// TIA Portal V17 export
// export: Created 2022-11-28T05:31:20.721325Z, ExportSetting WithDefaults, DisplayName Totally Integrated Automation Portal, DisplayVersion V17, DisplayName TIA Portal Openness, DisplayVersion V17, DisplayName TIA Portal Version Control Interface, DisplayVersion V17, DisplayName STEP 7 Professional, DisplayVersion V17, DisplayName STEP 7 Safety, DisplayVersion V17, DisplayName WinCC Professional, DisplayVersion V17
FUNCTION_BLOCK "FB_Sorting"   // FB1, LAD
{ S7_Optimized_Access := 'TRUE' }
VERSION : 0.1
// stored: AutoNumber true, IsIECCheckEnabled false, IsRetainMemResEnabled false, MemoryReserve 100, SetENOAutomatically false, UDAEnableTagReadback false
   VAR_INPUT
      Color : Int;
   END_VAR
   VAR
      "Step" : Int;
      IEC_Timer_Rojo { S7_SetPoint := 'True'} : TON_TIME;
      IEC_Timer_Eject { S7_SetPoint := 'True'} : TON_TIME;
      Detener_Banda { S7_SetPoint := 'True'} : TOF_TIME;
      Sensor_reading { S7_SetPoint := 'True'} : Int;
      IEC_Timer_ReadSensor { S7_SetPoint := 'True'} : TON_TIME;
      Conveyor0 { S7_SetPoint := 'True'} : Bool;
      Conveyor1 { S7_SetPoint := 'True'} : Bool;
      LapseEject : Time;
   END_VAR
   VAR CONSTANT
      LapseEjectWhite : Time := T#400ms;
      LapseEjectRed : Time := T#1400ms;
      LapseejectBlue : Time := T#2400ms;
   END_VAR
   VAR_TEMP   // added for the SCL form of the ladder/FBD networks
      _w1 : Bool;
   END_VAR
BEGIN

REGION Network 1
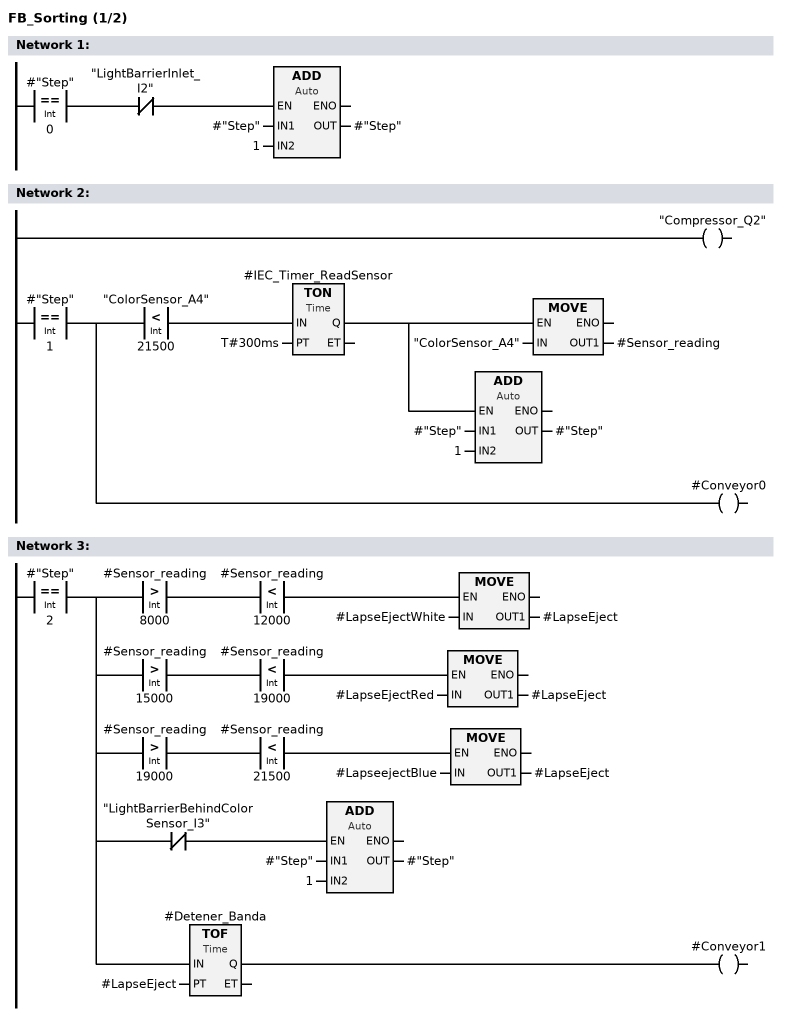
   RUNG wire#powerrail
      { S7_Templates := "SrcType := Int" } EQ_Contact(in1 := #"Step", in2 := 0)
      I_Contact( "LightBarrierInlet_I2" )
      Add(in1 := #"Step", in2 := 1, out => #"Step")
   END_RUNG
   // the same network as SCL:
   IF (#"Step" = 0) AND NOT "LightBarrierInlet_I2" THEN #"Step" := #"Step" + 1; END_IF;
END_REGION

REGION Network 2
   RUNG wire#powerrail
      Coil( "Compressor_Q2" )
   END_RUNG
   RUNG wire#powerrail
      { S7_Templates := "SrcType := Int" } EQ_Contact(in1 := #"Step", in2 := 1)
      wire#w1
      { S7_Templates := "SrcType := Int" } LT_Contact(in1 := "ColorSensor_A4", in2 := 21500)
      { S7_Templates := "time_type := Time" } #IEC_Timer_ReadSensor.TON(pt := T#300ms, et =>)
      wire#w2
      Move(in := "ColorSensor_A4", out1 => #Sensor_reading)
   END_RUNG
   RUNG wire#w2
      Add(in1 := #"Step", in2 := 1, out => #"Step")
   END_RUNG
   RUNG wire#w1
      Coil( #Conveyor0 )
   END_RUNG
   // the same network as SCL:
   "Compressor_Q2" := TRUE;
   #_w1 := #"Step" = 1;
   #IEC_Timer_ReadSensor(IN := #_w1 AND ("ColorSensor_A4" < 21500), PT := T#300ms);   // TON
   IF #IEC_Timer_ReadSensor.Q THEN
       #Sensor_reading := "ColorSensor_A4";
       #"Step" := #"Step" + 1;
   END_IF;
   #Conveyor0 := #_w1;
END_REGION

REGION Network 3
   RUNG wire#powerrail
      { S7_Templates := "SrcType := Int" } EQ_Contact(in1 := #"Step", in2 := 2)
      wire#w1
      { S7_Templates := "SrcType := Int" } GT_Contact(in1 := #Sensor_reading, in2 := 8000)
      { S7_Templates := "SrcType := Int" } LT_Contact(in1 := #Sensor_reading, in2 := 12000)
      Move(in := #LapseEjectWhite, out1 => #LapseEject)
   END_RUNG
   RUNG wire#w1
      { S7_Templates := "SrcType := Int" } GT_Contact(in1 := #Sensor_reading, in2 := 15000)
      { S7_Templates := "SrcType := Int" } LT_Contact(in1 := #Sensor_reading, in2 := 19000)
      Move(in := #LapseEjectRed, out1 => #LapseEject)
   END_RUNG
   RUNG wire#w1
      { S7_Templates := "SrcType := Int" } GT_Contact(in1 := #Sensor_reading, in2 := 19000)
      { S7_Templates := "SrcType := Int" } LT_Contact(in1 := #Sensor_reading, in2 := 21500)
      Move(in := #LapseejectBlue, out1 => #LapseEject)
   END_RUNG
   RUNG wire#w1
      I_Contact( "LightBarrierBehindColorSensor_I3" )
      Add(in1 := #"Step", in2 := 1, out => #"Step")
   END_RUNG
   RUNG wire#w1
      { S7_Templates := "time_type := Time" } #Detener_Banda.TOF(pt := #LapseEject, et =>)
      Coil( #Conveyor1 )
   END_RUNG
   // the same network as SCL:
   #_w1 := #"Step" = 2;
   IF #_w1 AND (#Sensor_reading > 8000) AND (#Sensor_reading < 12000) THEN
       #LapseEject := #LapseEjectWhite;
   END_IF;
   IF #_w1 AND (#Sensor_reading > 15000) AND (#Sensor_reading < 19000) THEN
       #LapseEject := #LapseEjectRed;
   END_IF;
   IF #_w1 AND (#Sensor_reading > 19000) AND (#Sensor_reading < 21500) THEN
       #LapseEject := #LapseejectBlue;
   END_IF;
   IF #_w1 AND NOT "LightBarrierBehindColorSensor_I3" THEN #"Step" := #"Step" + 1; END_IF;
   #Detener_Banda(IN := #_w1, PT := #LapseEject);   // TOF
   #Conveyor1 := #Detener_Banda.Q;
END_REGION

REGION Network 4
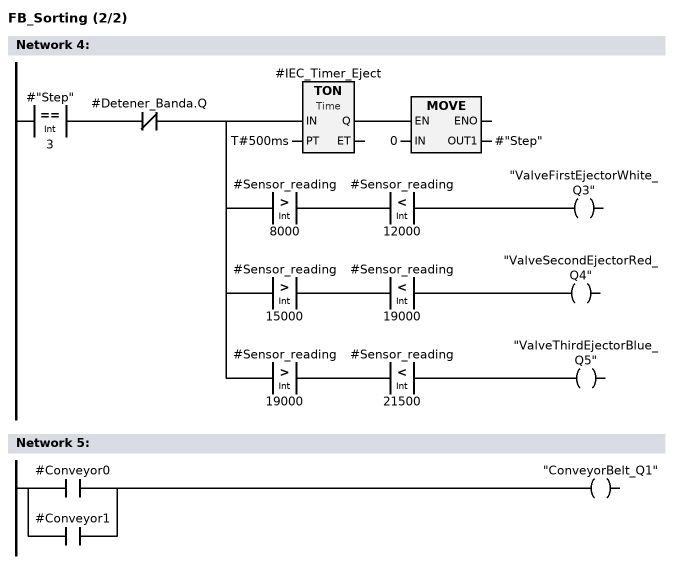
   RUNG wire#powerrail
      { S7_Templates := "SrcType := Int" } EQ_Contact(in1 := #"Step", in2 := 3)
      I_Contact( #Detener_Banda.Q )
      wire#w1
      { S7_Templates := "time_type := Time" } #IEC_Timer_Eject.TON(pt := T#500ms, et =>)
      Move(in := 0, out1 => #"Step")
   END_RUNG
   RUNG wire#w1
      { S7_Templates := "SrcType := Int" } GT_Contact(in1 := #Sensor_reading, in2 := 8000)
      { S7_Templates := "SrcType := Int" } LT_Contact(in1 := #Sensor_reading, in2 := 12000)
      Coil( "ValveFirstEjectorWhite_Q3" )
   END_RUNG
   RUNG wire#w1
      { S7_Templates := "SrcType := Int" } GT_Contact(in1 := #Sensor_reading, in2 := 15000)
      { S7_Templates := "SrcType := Int" } LT_Contact(in1 := #Sensor_reading, in2 := 19000)
      Coil( "ValveSecondEjectorRed_Q4" )
   END_RUNG
   RUNG wire#w1
      { S7_Templates := "SrcType := Int" } GT_Contact(in1 := #Sensor_reading, in2 := 19000)
      { S7_Templates := "SrcType := Int" } LT_Contact(in1 := #Sensor_reading, in2 := 21500)
      Coil( "ValveThirdEjectorBlue_Q5" )
   END_RUNG
   // the same network as SCL:
   #_w1 := (#"Step" = 3) AND NOT #Detener_Banda.Q;
   #IEC_Timer_Eject(IN := #_w1, PT := T#500ms);   // TON
   IF #IEC_Timer_Eject.Q THEN #"Step" := 0; END_IF;
   "ValveFirstEjectorWhite_Q3" := #_w1 AND (#Sensor_reading > 8000) AND (#Sensor_reading < 12000);
   "ValveSecondEjectorRed_Q4" := #_w1 AND (#Sensor_reading > 15000) AND (#Sensor_reading < 19000);
   "ValveThirdEjectorBlue_Q5" := #_w1 AND (#Sensor_reading > 19000) AND (#Sensor_reading < 21500);
END_REGION

REGION Network 5
   RUNG wire#powerrail
      Contact( #Conveyor0 )
      wire#w1
      Coil( "ConveyorBelt_Q1" )
   END_RUNG
   RUNG wire#powerrail
      Contact( #Conveyor1 )
   END_RUNG wire#w1
   // the same network as SCL:
   "ConveyorBelt_Q1" := #Conveyor0 OR #Conveyor1;
END_REGION
END_FUNCTION_BLOCK
